FUNCTION_BLOCK FB_AUT_130 EXTENDS FB_AUT_ABSTRACT
(****************************************************************************)
(*	POU_AUT_zxx			Bausteinaufrufe Station	zxx							*)
(*	Status				ungetestet											*)
(*  Version:			1.0													*)
(*	Beschrieb:																*)
(*																			*)
(*	Abläufe:			FB_ABLzxxA		Hauptablauf							*)
(*																			*)
(*																			*)
(* 	25.09.2019/Dj															*)
(****************************************************************************)
(*	dd.mm.yyyy   KZ    x.y			Beschrieb								*)
(****************************************************************************)
VAR_INPUT
    (* spezifische Eingänge *)

END_VAR
VAR_OUTPUT
    (* spezifische Ausgänge *)

END_VAR
VAR
    (* Bausteine *)
    fb_Dose : FB_ABL_130_Dose;

END_VAR

(*******************************************************************)
(* Timer *)
(*******************************************************************)

(*******************************************************************)
(* Flanken / Merker *)
(*******************************************************************)
//MANU CYCLE
IF (enIN_State = StateMANU) AND xIN_ManuCycle THEN
    xManuCycle := TRUE;
END_IF;

IF (enIN_State <> StateMANU) OR xOUT_Done THEN
    xManuCycle := FALSE;
END_IF

//NEXT STEP
xNextStep := (enIN_State > StateSTEP) OR
             ((enIN_State = StateSTEP) AND xIN_Step) OR
             ((enIN_State = StateMANU) AND xManuCycle);

//RESET
xReset := (enIN_State < StateREADY) AND (enIN_State <> StateINIT) AND NOT xManuCycle;

(*******************************************************************)
(* Bausteinaufrufe Abläufe *)
(*******************************************************************)

fb_Dose(xIN_Reset          := xReset,
       xIN_Init           := xIN_Init,
       xIN_Quit           := xIN_Quit,
       xIN_Start          := enIN_State = enState.StateAUTO, //AND _FB_ABL_100A.xOUT_Done AND _FB_ABL_100A.xOUT_Ready,
       xIN_Sperre         := NOT xIN_On,
       xIN_NextStep       := xNextStep,
       xIN_AlarmAktiv     := xIN_AlarmAktiv,
       xIN_DryCycle       := xIN_DryCycle,
       xIN_RestartCYCL    := enIN_State >= enState.StateLEER, // only restart when the mover has move out
       enIN_State         := enIN_State,
       tIN_Timeout        := tIN_Timeout,
       pxFG_Freigabe      := ADR(xDummy),
       Mover              := THIS^.Mover);

(*******************************************************************)
(* Mover reset flags *)
(*******************************************************************)

(*******************************************************************)
(* OUTPUT *)
(*******************************************************************)
xOUT_InitDone := fb_Dose.xOUT_InitDone;
xOUT_Ready    := fb_Dose.xOUT_Ready;
xOUT_Done     := fb_Dose.xOUT_Done;
xOUT_ErrFlag  := fb_Dose.xOUT_ErrFlag;
xOUT_Wait     := fb_Dose.xOUT_Wait;
xOUT_AlarmST  := xOUT_ErrFlag;

(*******************************************************************)
(* Bausteinaufruf Error Station *)
(*******************************************************************)
// POU_ERR_VORLAGE(xIN_QUIT:=xIN_Quit , pstrArIN_ALARM:=ADR(HMI.strArALARM[1]));

(* % of completion of the process *)
PROPERTY iCompletionPC : INT
GET
iCompletionPC := THIS^.fb_Dose.iOUT_ProcessCompletion;
END_GET
END_PROPERTY

PROPERTY ProcessExecution : ProcessExecution_e
GET
ProcessExecution := THIS^._ProcessExecution;
END_GET
SET
THIS^._ProcessExecution := ProcessExecution;
END_SET
END_PROPERTY

PROPERTY xBusy : BOOL
GET
xBusy := THIS^.fb_Dose.xOUT_Busy;
END_GET
SET
END_SET
END_PROPERTY

PROPERTY xDone : BOOL
GET
xDone := THIS^.fb_Dose.xOUT_Ready OR THIS^.fb_Dose.xOUT_Done;
END_GET
END_PROPERTY

PROPERTY xMoverPathFree : BOOL
GET
xMoverPathFree := THIS^.fb_Dose.xOUT_MoverFree OR THIS^.fb_Dose.xOUT_Ready OR THIS^.fb_Dose.xOUT_Done;
END_GET
END_PROPERTY

PROPERTY xMoverShouldLeave : BOOL
GET
xMoverShouldLeave := THIS^.fb_Dose.iOUT_Step = ST130_Dose_e.SYNC_MOVER_LEAVE;
END_GET
END_PROPERTY

END_FUNCTION_BLOCK

(* stored: Version 1.1.0.1, ProductVersion 3.1.4024.6
   POU FB_AUT_130: Id {aabc6712-002c-446d-a55f-42f6063f8dd2}, SpecialFunc None
   Property iCompletionPC: Id {a6312a84-bdfa-44ce-8e04-c9e231e2340c}
   Get Get: Id {68ad4865-5843-4968-9afb-1ed0fc0d671f}
   Property ProcessExecution: Id {d87c4446-298f-49bd-be30-3867757bc7eb}
   Get Get: Id {ecf337d4-2712-419b-ad0b-e0ca1057b401}
   Set Set: Id {689f384d-3307-4429-b6ea-0a70259f8823}
   Property xBusy: Id {d7403fc9-ab79-40a2-b205-fdd7afb85837}
   Get Get: Id {8d8117ef-acf2-4a79-bfa3-f4beee5a809b}
   Set Set: Id {8a417c9c-b913-4c95-b965-485fa973e661}
   Property xDone: Id {151d7923-ba15-4380-96a6-a22c27ea74e0}
   Get Get: Id {8c05b73b-594a-4c39-af60-b2a891e3b0cc}
   Property xMoverPathFree: Id {72c8ed4a-52c7-4268-8661-42711cbe97bb}
   Get Get: Id {0de9805a-be8f-4322-a342-e80cba055a76}
   Property xMoverShouldLeave: Id {cc9a3f79-f20e-4845-acf0-98e6bde159cb}
   Get Get: Id {3d3e22a4-131b-468d-b0c9-59c2cfe06f9a} *)
